FUNCTION_BLOCK FB_Nagel
VAR_INPUT
	visible:BOOL;
END_VAR

END_FUNCTION_BLOCK

(* stored: Version 1.1.0.1, ProductVersion 3.1.4024.3
   POU FB_Nagel: Id {bf58f65c-449f-41ac-9910-73b494142a45}, SpecialFunc None *)
